(* CoDeSys 2.3 export: ST_CAN_NODESTATE.EXP *)

(* Data type *)
TYPE ST_CAN_NODESTATE :
STRUCT
	Desc : STRING;

	(*Alarm*)
	Alarm  : ST_ALARM;

END_STRUCT
END_TYPE
